(* CODESYS project SistemaBombasGabrielPedro.project

Project tree, tasks and I/O mapping:
  Device : CODESYS Control Win V3, 3S - Smart Software Solutions GmbH, order no. 305021, version 3.5.11.40
    application Application
      libraries: Standard, * (System)
      task MainTask (cyclic, interval t#20ms, priority 1) calls FUEL_PUMPING
      program FUEL_PUMPING [ST]
      global variables GVL
      Docks/
        Automatic/
          program Doca1_auto [SFC]
          program Doca2_auto [ST]
        Manual/
      Simulation/
        Automatic/
          program Doca1_Simulation_Auto [ST]
          program Doca2_Simulation_Auto [ST]
*)

// Device/Application/GVL
{attribute 'qualified_only'}
VAR_GLOBAL   
	Y_C_D1, Y_C_D2: BOOL;         (* Presença de caminhões nas docas *)
    Y_M_D1, Y_M_D2: BOOL;         (* Mangueiras acopladas *)
    LSH_S01, LSH_S02, LSH_S03: BOOL; (* Nível alto dos silos *)
    LSL_S01, LSL_S02, LSL_S03: BOOL; (* Nível baixo dos silos *)
    LT_S01, LT_S02, LT_S03: REAL; (* Nível contínuo dos silos *)
    BOTAO_EMERGENCIA: BOOL;       (* Botão de emergência *)
	
	VA_S01, VA_S02, VA_S03: BOOL; (* Válvulas de admissão *)
    VS_S01, VS_S02_1, VS_S02_2, VS_S03, VC_TQ1, VC_TQ2: BOOL; (* Válvulas de saída *)
    B_R1, B_R2: BOOL;             (* Bombas *)
    M1, M2: BOOL;                 (* Motores de agitação *)
    C_D1, C_D2: BOOL;             (* Cancelas das docas *)
    ESTADO_EMERGENCIA: BOOL;      (* Estado do sistema em emergência *)
	
	
	
	ESTADO_DOCA1, ESTADO_DOCA2: INT; (* Estado das sequências nas docas *)
    VOLUME_CARREGADO_D1, VOLUME_CARREGADO_D2: REAL; (* Volume carregado *)
    CAPACIDADE_CAMINHAO: REAL := 25000;       (* Capacidade máxima do caminhão *)
	caminhao1_cheio: BOOL := FALSE;
	caminhao2_cheio: BOOL :=FALSE;
    VAZAO_CARREGAMENTO: REAL := 500.0; (* Vazão de carregamento em litros/s *)
    TempoCiclo: REAL := 0.01;         (* Tempo de ciclo do programa em segundos *)
    INIT: BOOL := FALSE;             (* Variável de inicialização *)
	
	
	ALARME_NIVEL_ALTO_S01, ALARME_NIVEL_BAIXO_S01: BOOL;
    ALARME_NIVEL_ALTO_S02, ALARME_NIVEL_BAIXO_S02: BOOL;
    ALARME_NIVEL_ALTO_S03, ALARME_NIVEL_BAIXO_S03: BOOL;
	EMERGENCIA: BOOL;
	
	VOLUME_S01, VOLUME_S02, VOLUME_S03: REAL; (* Volumes dos silos *)
    VOLUME_TQ1, VOLUME_TQ2: REAL;            (* Volumes dos tanques *)
    VOLUME_R1, VOLUME_R2: REAL := 250000;    (* Volumes dos reservatórios *)
    CAPACIDADE_SILO: REAL := 50000.0;        (* Capacidade dos silos *)
    CAPACIDADE_TQ: REAL := 25000.0;          (* Capacidade dos tanques de mistura *)
    CAPACIDADE_RESERVATORIO: REAL := 250000.0; (* Capacidade dos reservatórios *)
	GAS_TYPE: INT := -1; (* Tipo de gasolina selecionado pelo operador, 0 para etanol, 1 para comum, 2 para premium *)
	MIXER_TIMER: TON;
	
	
	
	
END_VAR

// Device/Application/FUEL_PUMPING
PROGRAM FUEL_PUMPING

(* Variáveis internas *)
VAR
    MODO_AUTOMATICO: BOOL := TRUE; (* Ativar modo automático por padrão *)
    TempoCiclo: REAL := 0.1;       (* Tempo de ciclo do programa em segundos *)
END_VAR

(* Lógica de alternância de modos *)
IF MODO_AUTOMATICO THEN
    (* Chamar os blocos automáticos das docas *)
    Doca1_auto();
    Doca2_auto();

    (* Simulação dos modos automáticos para as docas *)
    Doca1_Simulation_Auto();
    Doca2_Simulation_Auto();
ELSE
    (* Caso nenhum modo esteja ativo, desligar tudo *)
    GVL.VA_S01 := FALSE;
    GVL.VA_S02 := FALSE;
    GVL.VA_S03 := FALSE;

    GVL.VS_S01 := FALSE;
    GVL.VS_S02_1 := FALSE;
    GVL.VS_S02_2 := FALSE;
    GVL.VS_S03 := FALSE;

    GVL.B_R1 := FALSE;
    GVL.B_R2 := FALSE;

    GVL.M1 := FALSE;
    GVL.M2 := FALSE;
END_IF;

(* Tratamento de Emergência *)
IF GVL.BOTAO_EMERGENCIA THEN
    (* Interromper todas as operações *)
    GVL.VA_S01 := FALSE;
    GVL.VA_S02 := FALSE;
    GVL.VA_S03 := FALSE;

    GVL.VS_S01 := FALSE;
    GVL.VS_S02_1 := FALSE;
    GVL.VS_S02_2 := FALSE;
    GVL.VS_S03 := FALSE;

    GVL.B_R1 := FALSE;
    GVL.B_R2 := FALSE;

    GVL.M1 := FALSE;
    GVL.M2 := FALSE;

    GVL.C_D1 := FALSE;
    GVL.C_D2 := FALSE;

    GVL.ESTADO_EMERGENCIA := TRUE;
ELSE
    GVL.ESTADO_EMERGENCIA := FALSE;
END_IF;

END_PROGRAM

// Device/Application/Docks/Automatic/Doca1_auto
PROGRAM Doca1_auto
VAR_INPUT
	GAS_FILL: BOOL;
	ETA_FILL: BOOL;
END_VAR

VAR
	ESTADO_DOCA1: INT := 0;
	COUNTER: INT := 0;
END_VAR

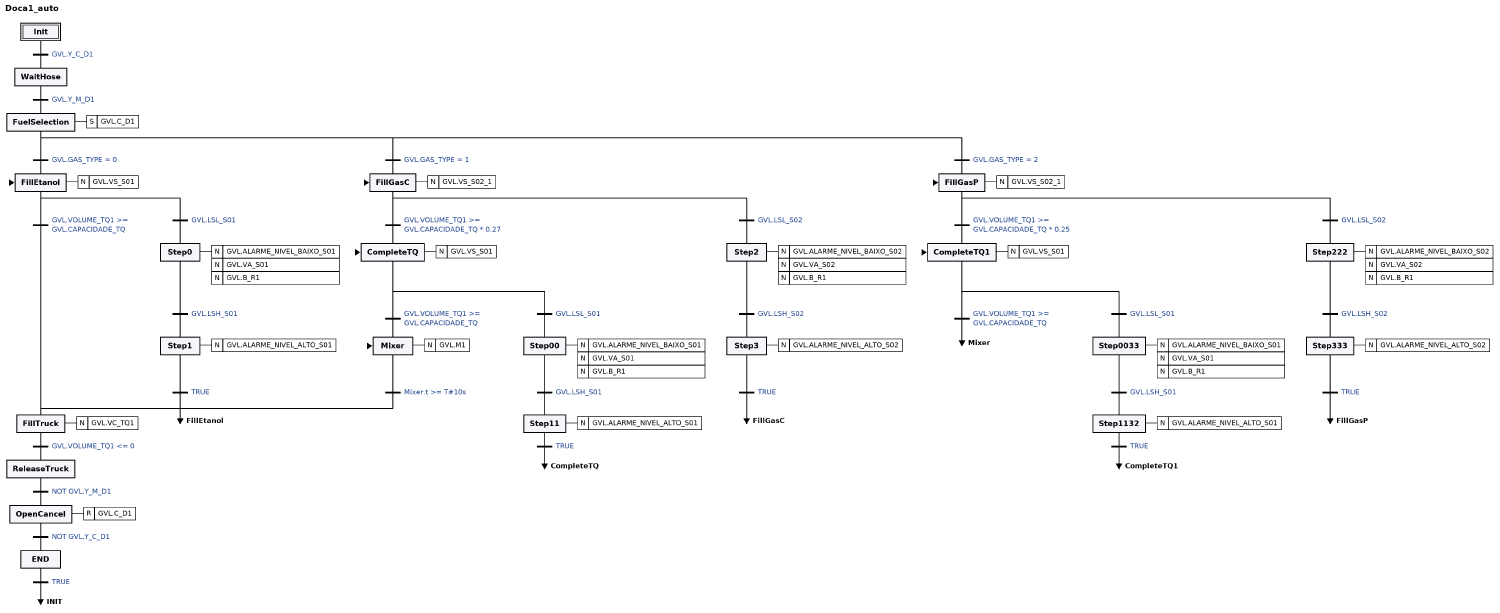
INITIAL_STEP Init:
END_STEP
TRANSITION FROM Init TO WaitHose
    := GVL.Y_C_D1;
END_TRANSITION
STEP WaitHose:
END_STEP
TRANSITION FROM WaitHose TO FuelSelection
    := GVL.Y_M_D1;
END_TRANSITION
STEP FuelSelection:
    GVL.C_D1(S);
END_STEP
TRANSITION FROM FuelSelection TO FillEtanol
    := GVL.GAS_TYPE = 0;
END_TRANSITION
STEP FillEtanol:
    GVL.VS_S01(N);
END_STEP
TRANSITION FROM FillEtanol TO FillTruck
    := GVL.VOLUME_TQ1 >= GVL.CAPACIDADE_TQ;
END_TRANSITION
TRANSITION FROM FillEtanol TO Step0
    := GVL.LSL_S01;
END_TRANSITION
STEP Step0:
    GVL.ALARME_NIVEL_BAIXO_S01(N);
    GVL.VA_S01(N);
    GVL.B_R1(N);
END_STEP
TRANSITION FROM Step0 TO Step1
    := GVL.LSH_S01;
END_TRANSITION
STEP Step1:
    GVL.ALARME_NIVEL_ALTO_S01(N);
END_STEP
TRANSITION FROM Step1 TO FillEtanol
    := TRUE;
END_TRANSITION
TRANSITION FROM FuelSelection TO FillGasC
    := GVL.GAS_TYPE = 1;
END_TRANSITION
STEP FillGasC:
    GVL.VS_S02_1(N);
END_STEP
TRANSITION FROM FillGasC TO CompleteTQ
    := GVL.VOLUME_TQ1 >= GVL.CAPACIDADE_TQ * 0.27;
END_TRANSITION
TRANSITION FROM FillGasC TO Step2
    := GVL.LSL_S02;
END_TRANSITION
STEP Step2:
    GVL.ALARME_NIVEL_BAIXO_S02(N);
    GVL.VA_S02(N);
    GVL.B_R1(N);
END_STEP
TRANSITION FROM Step2 TO Step3
    := GVL.LSH_S02;
END_TRANSITION
STEP Step3:
    GVL.ALARME_NIVEL_ALTO_S02(N);
END_STEP
TRANSITION FROM Step3 TO FillGasC
    := TRUE;
END_TRANSITION
STEP CompleteTQ:
    GVL.VS_S01(N);
END_STEP
TRANSITION FROM CompleteTQ TO Mixer
    := GVL.VOLUME_TQ1 >= GVL.CAPACIDADE_TQ;
END_TRANSITION
TRANSITION FROM CompleteTQ TO Step00
    := GVL.LSL_S01;
END_TRANSITION
STEP Step00:
    GVL.ALARME_NIVEL_BAIXO_S01(N);
    GVL.VA_S01(N);
    GVL.B_R1(N);
END_STEP
TRANSITION FROM Step00 TO Step11
    := GVL.LSH_S01;
END_TRANSITION
STEP Step11:
    GVL.ALARME_NIVEL_ALTO_S01(N);
END_STEP
TRANSITION FROM Step11 TO CompleteTQ
    := TRUE;
END_TRANSITION
STEP Mixer:
    GVL.M1(N);
END_STEP
TRANSITION FROM Mixer TO FillTruck
    := Mixer.t >= T#10s;
END_TRANSITION
TRANSITION FROM FuelSelection TO FillGasP
    := GVL.GAS_TYPE = 2;
END_TRANSITION
STEP FillGasP:
    GVL.VS_S02_1(N);
END_STEP
TRANSITION FROM FillGasP TO CompleteTQ1
    := GVL.VOLUME_TQ1 >= GVL.CAPACIDADE_TQ * 0.25;
END_TRANSITION
STEP CompleteTQ1:
    GVL.VS_S01(N);
END_STEP
TRANSITION FROM FillGasP TO Step222
    := GVL.LSL_S02;
END_TRANSITION
STEP Step222:
    GVL.ALARME_NIVEL_BAIXO_S02(N);
    GVL.VA_S02(N);
    GVL.B_R1(N);
END_STEP
TRANSITION FROM Step222 TO Step333
    := GVL.LSH_S02;
END_TRANSITION
STEP Step333:
    GVL.ALARME_NIVEL_ALTO_S02(N);
END_STEP
TRANSITION FROM Step333 TO FillGasP
    := TRUE;
END_TRANSITION
TRANSITION FROM CompleteTQ1 TO Mixer
    := GVL.VOLUME_TQ1 >= GVL.CAPACIDADE_TQ;
END_TRANSITION
TRANSITION FROM CompleteTQ1 TO Step0033
    := GVL.LSL_S01;
END_TRANSITION
STEP Step0033:
    GVL.ALARME_NIVEL_BAIXO_S01(N);
    GVL.VA_S01(N);
    GVL.B_R1(N);
END_STEP
TRANSITION FROM Step0033 TO Step1132
    := GVL.LSH_S01;
END_TRANSITION
STEP Step1132:
    GVL.ALARME_NIVEL_ALTO_S01(N);
END_STEP
TRANSITION FROM Step1132 TO CompleteTQ1
    := TRUE;
END_TRANSITION
STEP FillTruck:
    GVL.VC_TQ1(N);
END_STEP
TRANSITION FROM FillTruck TO ReleaseTruck
    := GVL.VOLUME_TQ1 <= 0;
END_TRANSITION
STEP ReleaseTruck:
END_STEP
TRANSITION FROM ReleaseTruck TO OpenCancel
    := NOT GVL.Y_M_D1;
END_TRANSITION
STEP OpenCancel:
    GVL.C_D1(R);
END_STEP
TRANSITION FROM OpenCancel TO END
    := NOT GVL.Y_C_D1;
END_TRANSITION
STEP END:
END_STEP
TRANSITION FROM END TO INIT
    := TRUE;
END_TRANSITION

END_PROGRAM

// Device/Application/Docks/Automatic/Doca2_auto
PROGRAM Doca2_auto
VAR_INPUT
    GAS_FILL: BOOL;
    ETA_FILL: BOOL;
END_VAR

VAR
    ESTADO_DOCA2: INT := 0;
END_VAR

(* Lógica da Doca 2 no Modo Automático *)
CASE ESTADO_DOCA2 OF

    0: (* Aguardando Caminhão *)
        IF GVL.Y_C_D2 THEN
            ESTADO_DOCA2 := 1; (* Caminhão detectado, próximo estado *)
        END_IF;

    1: (* Verificar Conexão da Mangueira *)
        IF GVL.Y_M_D2 THEN
            GVL.C_D2 := TRUE; (* Fechar a cancela *)
            ESTADO_DOCA2 := 2; (* Passar para o próximo estado *)
        END_IF;

    2: (* Seleção do Combustível *)
        IF GAS_FILL THEN
            ESTADO_DOCA2 := 3; (* Gasolina selecionada *)
        ELSIF ETA_FILL THEN
            ESTADO_DOCA2 := 4; (* Etanol selecionado *)
        END_IF;

    3: (* Carregamento de Gasolina *)
        GVL.VS_S02_2 := TRUE; (* Abrir válvula de saída do silo S02 para TQ2 *)
        GVL.B_R2 := TRUE;     (* Ativar bomba de gasolina *)

        (* Controle de volume *)
        IF GVL.VOLUME_CARREGADO_D2 >= GVL.CAPACIDADE_CAMINHAO THEN
            GVL.VS_S02_2 := FALSE; (* Fechar válvula de saída *)
            GVL.B_R2 := FALSE;     (* Desligar bomba *)
            ESTADO_DOCA2 := 5;     (* Carregamento concluído *)
        END_IF;

    4: (* Carregamento de Etanol *)
        GVL.VS_S03 := TRUE; (* Abrir válvula de saída do silo S03 *)
        GVL.B_R1 := TRUE;   (* Ativar bomba de etanol *)

        (* Controle de volume *)
        IF GVL.VOLUME_CARREGADO_D2 >= GVL.CAPACIDADE_CAMINHAO THEN
            GVL.VS_S03 := FALSE; (* Fechar válvula de saída *)
            GVL.B_R1 := FALSE;   (* Desligar bomba *)
            ESTADO_DOCA2 := 5;   (* Carregamento concluído *)
        END_IF;

    5: (* Finalizando Carregamento *)
        IF NOT GVL.Y_M_D2 THEN
            GVL.C_D2 := FALSE; (* Abrir a cancela para liberar o caminhão *)
            ESTADO_DOCA2 := 6;   (* Caminhão pode sair *)
        END_IF;

    6: (* Aguardando Saída do Caminhão *)
        IF NOT GVL.Y_C_D2 THEN
            ESTADO_DOCA2 := 0; (* Caminhão saiu, reinicia o processo *)
        END_IF;

    ELSE
        ESTADO_DOCA2 := 0; (* Estado inválido, reinicia *)
END_CASE;

(* Monitoramento de Níveis Críticos *)
IF GVL.LSL_S03 THEN
    GVL.ALARME_NIVEL_BAIXO_S03 := TRUE;
END_IF;

IF GVL.LSH_S03 THEN
    GVL.ALARME_NIVEL_ALTO_S03 := TRUE;
END_IF;

IF GVL.LSL_S02 THEN
    GVL.ALARME_NIVEL_BAIXO_S02 := TRUE;
END_IF;

IF GVL.LSH_S02 THEN
    GVL.ALARME_NIVEL_ALTO_S02 := TRUE;
END_IF;

(* Tratamento de Emergência *)
IF GVL.BOTAO_EMERGENCIA THEN
    GVL.C_D2 := FALSE; (* Liberar a cancela *)
    GVL.VS_S03 := FALSE;
    GVL.VS_S02_2 := FALSE;
    GVL.B_R1 := FALSE;
    GVL.B_R2 := FALSE;
    ESTADO_DOCA2 := 0; (* Reinicia o processo *)
END_IF;

END_PROGRAM

// Device/Application/Simulation/Automatic/Doca1_Simulation_Auto
PROGRAM Doca1_Simulation_Auto
VAR
    TempoCiclo: REAL := 1; (* Tempo de ciclo do programa em segundos *)
END_VAR

(* Atualizar sensores de nível do silo S01 *)
IF GVL.volume_S01 <= (GVL.CAPACIDADE_SILO * 0.1) THEN
	GVL.LSL_S01 := TRUE;
ELSE
	GVL.LSL_S01 := FALSE;
END_IF;

IF GVL.volume_S01 >= (GVL.CAPACIDADE_SILO * 0.9) THEN
	GVL.LSH_S01 := TRUE;
ELSE
	GVL.LSH_S01 := FALSE;
END_IF;

(*Encher o tanque 1 de etanol*)
IF GVL.VS_S01 AND NOT GVL.LSL_S01 THEN
	IF GVL.VOLUME_S01 > 0 AND NOT (GVL.VOLUME_TQ1 > GVL.CAPACIDADE_TQ) THEN
        GVL.VOLUME_S01 := GVL.VOLUME_S01 - (GVL.VAZAO_CARREGAMENTO * TempoCiclo);
        GVL.VOLUME_TQ1 := GVL.VOLUME_TQ1 + (GVL.VAZAO_CARREGAMENTO * TempoCiclo);
    END_IF;

END_IF

(*Encher o tanque 1 de Gasolina*)
IF GVL.VS_S02_1 AND NOT GVL.LSL_S02 THEN
	IF GVL.VOLUME_S02 > 0 AND NOT (GVL.VOLUME_TQ1 > GVL.CAPACIDADE_TQ) THEN
		GVL.VOLUME_S02 := GVL.VOLUME_S02 - (GVL.VAZAO_CARREGAMENTO * TempoCiclo);
		GVL.VOLUME_TQ1 := GVL.VOLUME_TQ1 + ( GVL.VAZAO_CARREGAMENTO * TempoCiclo);
		END_IF
	END_IF

(*Encher o caminhão doca 1*)
IF GVL.VC_TQ1 THEN
	IF GVL.VOLUME_TQ1 > 0  THEN
        GVL.VOLUME_TQ1 := GVL.VOLUME_TQ1 - (GVL.VAZAO_CARREGAMENTO * TempoCiclo);
        GVL.VOLUME_CARREGADO_D1 := GVL.VOLUME_CARREGADO_D1 + (GVL.VAZAO_CARREGAMENTO * TempoCiclo);
    END_IF;
END_IF

IF NOT GVL.LSH_S01 AND GVL.B_R1 AND GVL.VA_S01 THEN
	IF GVL.VOLUME_R1 > 0 THEN
		GVL.VOLUME_R1 := GVL.VOLUME_R1 - (GVL.VAZAO_CARREGAMENTO * TempoCiclo);
		GVL.VOLUME_S01 := GVL.VOLUME_S01 + (GVL.VAZAO_CARREGAMENTO * TempoCiclo);
	END_IF
END_IF

END_PROGRAM

// Device/Application/Simulation/Automatic/Doca2_Simulation_Auto
PROGRAM Doca2_Simulation_Auto
VAR
    TempoCiclo: REAL := 5; (* Tempo de ciclo do programa em segundos *)
END_VAR

(* Lógica de Simulação *)

(* Simulação do comportamento do Silo S03 *)
IF GVL.VS_S03 AND GVL.Y_C_D2 THEN
    (* Esvaziando o Silo S03 para o caminhão *)
    IF GVL.volume_S03 > 0 THEN
        GVL.volume_S03 := GVL.volume_S03 - (GVL.VAZAO_CARREGAMENTO * TempoCiclo);
        GVL.VOLUME_CARREGADO_D2 := GVL.VOLUME_CARREGADO_D2 + (GVL.VAZAO_CARREGAMENTO * TempoCiclo);
    END_IF;

    (* Atualizar sensores de nível do silo S03 *)
    IF GVL.volume_S03 <= (GVL.CAPACIDADE_SILO * 0.1) THEN
        GVL.LSL_S03 := TRUE;
    ELSE
        GVL.LSL_S03 := FALSE;
    END_IF;

    IF GVL.volume_S03 >= (GVL.CAPACIDADE_SILO * 0.9) THEN
        GVL.LSH_S03 := TRUE;
    ELSE
        GVL.LSH_S03 := FALSE;
    END_IF;
END_IF;

(* Simulação do comportamento do Silo S02 *)
IF GVL.VS_S02_2 AND GVL.Y_C_D2 THEN
    (* Esvaziando o Silo S02 para o tanque TQ2 *)
    IF GVL.volume_S02 > 0 THEN
        GVL.volume_S02 := GVL.volume_S02 - (GVL.VAZAO_CARREGAMENTO * TempoCiclo);
        GVL.VOLUME_CARREGADO_D2 := GVL.VOLUME_CARREGADO_D2 + (GVL.VAZAO_CARREGAMENTO * TempoCiclo);
    END_IF;

    (* Atualizar sensores de nível do silo S02 *)
    IF GVL.volume_S02 <= (GVL.CAPACIDADE_SILO * 0.1) THEN
        GVL.LSL_S02 := TRUE;
    ELSE
        GVL.LSL_S02 := FALSE;
    END_IF;

    IF GVL.volume_S02 >= (GVL.CAPACIDADE_SILO * 0.9) THEN
        GVL.LSH_S02 := TRUE;
    ELSE
        GVL.LSH_S02 := FALSE;
    END_IF;
END_IF;

(* Simulação do comportamento do Tanque TQ2 *)
IF GVL.VOLUME_CARREGADO_D2 >= GVL.CAPACIDADE_CAMINHAO THEN
    (* Caminhão cheio *)
    GVL.caminhao2_cheio := TRUE;
    GVL.VS_S03 := FALSE;
    GVL.VS_S02_2 := FALSE;
ELSE
    GVL.caminhao2_cheio := FALSE;
END_IF;

(* Tratamento de Emergência *)
IF GVL.EMERGENCIA THEN
    (* Interromper todas as operações *)
    GVL.VS_S03 := FALSE;
    GVL.VS_S02_2 := FALSE;
    GVL.B_R1 := FALSE;
    GVL.B_R2 := FALSE;

    (* Reiniciar volumes *)
    GVL.VOLUME_CARREGADO_D2 := 0;
    GVL.caminhao2_cheio := FALSE;
END_IF;

END_PROGRAM
